Universal Robots PolyScope program: passatronko2.urp

Program passatronko2 (installation=default directory=/programs createdIn=3.10.1.76190 lastSavedIn=5.9.3.1031212 robotSerialNumber=20195300809)
Calibrated DH parameters: a=[-0.000085, -0.20076, -0.212369, 0.000121, -0.000118, 0]; d=[0.15185, -26.306375, 24.753047, 1.684739, 0.085386, 0.092088]; alpha=[1.572149, -0.00522, -0.011864, 1.571339, -1.571085, 0]; deltaTheta=[0, 0.599885, -0.513355, -0.086555, 0.000006, 0]
BeforeStart
  con := socket_open("10.5.20.90",30002)
Robot Program (runOnlyOnce=false)
  Loop While (checkContinuously=false) expression=con≟ True
    con := socket_open("10.5.20.90",30002)
    Popup Message (haltProgram=false message=hola inputType=Text)
    Wait Sleep waitTime=0.01
    str := "Passa tronco"
    Script: socket_send_string(str)
    Script: socket_send_byte(10)
    Script: socket_close()
